FUNCTION WRITE_ANY_BYTE : BOOL
VAR_INPUT
    ptr: POINTER TO BYTE;
    val: BYTE;
END_VAR

ptr^ := val;

END_FUNCTION

(* stored: Version 1.1.0.1, ProductVersion 3.1.4022.9
   POU WRITE_ANY_BYTE: Id {0bd58fcc-2342-4cd5-b054-08bdfb22baa1}, SpecialFunc None *)
